RoboDK station: RoboDK Project-Station Kawasaki BA006L.rdk

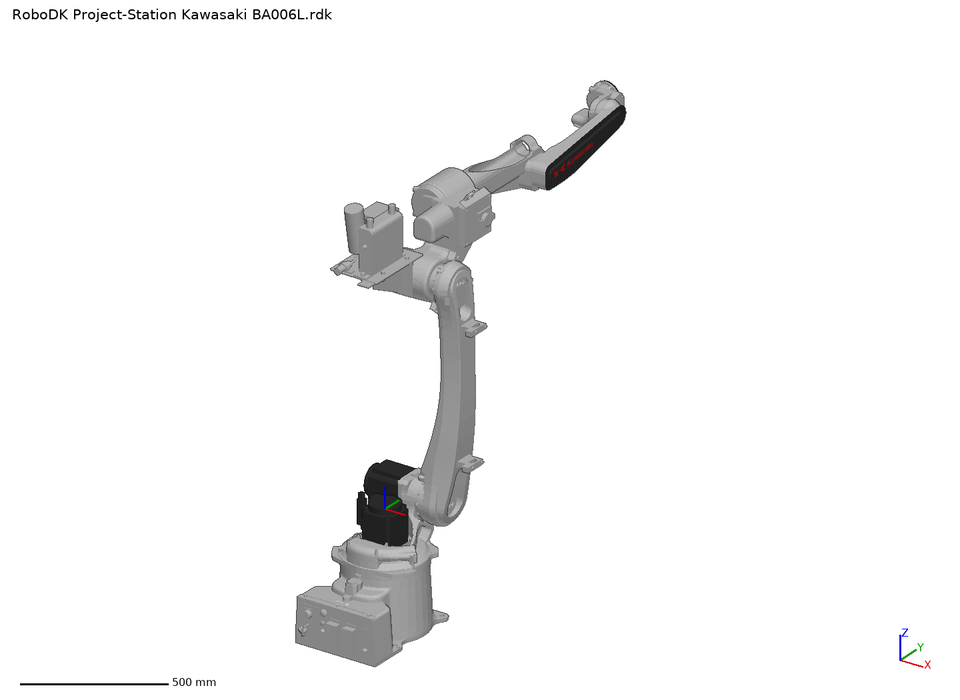
[picture v0: the station drawn from its stored meshes, robots at their saved joint values, targets as dots, program paths as lines]
Station Station Kawasaki BA006L (saved by RoboDK 5.6.4). Poses are relative to the parent item; angles as X-Y-Z fixed-axis rotations.
Station parameters (name, value as stored): WASM
  - frame Kawasaki BA006L Base at (0, 0, 430) mm
    - robot Kawasaki BA006L: 6 axes, payload 6 kg, reach 2036 mm, repeatability 0.08 mm, weight 160 kg
        modified DH rows (alpha deg, a mm, theta deg, d mm): 0, 0, 0, 430; -90, 165, -90, 0; 0, 820, -90, 0; -90, 210, 0, 1030; 90, 0, 0, 0; -90, 0, 180, 115
        base shift (0, 0, -430) mm, rotated rx 0 ry 0 rz 90 deg
        joint limits [-165, -90, -155, -180, -135, -360] to [165, 150, 135, 180, 135, 360]; home [0, 0, -90, 0, 0, 0]; saved at [0, 0, -90, 0, 0, 0]
